# EPICS substitutions: te_tc/te_tcApp/Db/te_tc.substitutions
file te_tc.template { pattern
{ Sys	, Dev		,PORT		, Chan	}
{ Depo	, "{TC:1}"	, Depo_TC1	, 1	}
}
